TYPE TTransferIndex :
	(TI_Loader:=0,TI_LoaderTableL1,TI_LoaderTableL2,TI_LoaderTableR1,TI_LoaderTableR2,TI_PearlingTableL,TI_PearlingTableR,TI_PearlingTable, TI_LoaderTurnOver,TI_END);
END_TYPE

(* stored: Version 1.1.0.1, ProductVersion 3.1.4022.12
   DUT TTransferIndex: Id {0c80fbdd-108b-4184-9476-11d2c7125670} *)
